PROGRAM Fast_Faults
VAR
END_VAR

g_FastFaultOutput1();

END_PROGRAM

(* stored: Version 1.1.0.1, ProductVersion 3.1.4022.12
   POU Fast_Faults: Id {bdc9fda1-3ab8-0d1a-09bd-274a15fdc835}, SpecialFunc None *)
